// TIA Portal V16 export
// export: Created 2022-11-17T15:49:44.5992417Z, ExportSetting WithDefaults, DisplayName Totally Integrated Automation Portal, DisplayVersion V16 Update 6, DisplayName TIA Portal Version Control Interface, DisplayVersion V16 Update 2, DisplayName TIA Portal Openness, DisplayVersion V16 Update 6, DisplayName SINAMICS Startdrive Advanced, DisplayVersion V16 Update 5, DisplayName SINAMICS Startdrive G130, G150, S120, S150, SINAMICS MV, S210, DisplayVersion V16 Update 5, DisplayName SINAMICS Startdrive G110M, G120, G120C, G120D, G120P, G115D, DisplayVersion V16 Update 5, DisplayName STEP 7 Professional, DisplayVersion V16 Update 6, DisplayName STEP 7 Safety, DisplayVersion V16, DisplayName WinCC Advanced, DisplayVersion V16 Update 6
DATA_BLOCK "DB241_Program9"   // DB241
{ S7_Optimized_Access := 'FALSE' }
AUTHOR : Robopac
VERSION : 0.0
// stored: AutoNumber false, IsOnlyStoredInLoadMemory false, IsWriteProtectedInAS false
   VAR RETAIN
      Program9 { S7_SetPoint := 'True'} : "DatiProgramma";
   END_VAR
BEGIN
   Program9.Wrapping := TRUE;
   Program9.TopLenght := 500;
   Program9.TopRelease := 0;
   Program9.TopDown := 0;
   Program9.Top := 4;
   Program9.PressurePTime := 0;
   Program9.LifterTime := 0;
   Program9.RevOverContrast := 1;
   Program9.RopeEndCycle := 16#02;
   Program9.Spare4 := 16#01;
   Program9.RopeTime := 1500;
   Program9.RevOverClamp := 1;
   Program9.FilmForceFinalRev := 10;
   Program9.FilmPrestretchFinalRev := 100;
   Program9.ArmSpeed := 100;
   Program9.CarriageDown4Top := 500;
   Program9.TopDownTime := 1500;
   Program9.LapsUnderTop := 0;
   Program9.Spare6 := 0;
   Program9.Spare7 := 0;
   Program9.Spare8 := 0;
   Program9.Spare9 := 0;
   Program9.Spare10 := 0;
   Program9.Spare11 := 0;
   Program9.Spare12 := 0;
   Program9.Overlap0_1 := 0;
   Program9.Height1 := 130;
   Program9.Landmark1 := FALSE;
   Program9.Lifter1 := FALSE;
   Program9.SpareBit1H1 := FALSE;
   Program9.Airblower1 := TRUE;
   Program9.NextStep1 := TRUE;
   Program9.PressureP1 := TRUE;
   Program9.SpareByte2H1 := 16#00;
   Program9.Revolution1 := 1;
   Program9.RopeUnit1_1 := 16#01;
   Program9.RopeUnit1_2 := 16#01;
   Program9.FilmForce1 := 5;
   Program9.FilmPrestretch1 := 200;
   Program9.Spare3H1 := 0;
   Program9.Spare49 := 0;
   Program9.Spare50 := 0;
   Program9.Spare51 := 0;
   Program9.Spare52 := 0;
   Program9.Spare53 := 0;
   Program9.Overlap1_2 := 0;
   Program9.Height2 := 50;
   Program9.Landmark2 := FALSE;
   Program9.Lifter2 := FALSE;
   Program9.SpareBit1H2 := FALSE;
   Program9.Airblower2 := TRUE;
   Program9.NextStep2 := TRUE;
   Program9.PressureP2 := TRUE;
   Program9.SpareByte2H2 := 16#00;
   Program9.Revolution2 := 1;
   Program9.RopeUnit2_1 := 16#01;
   Program9.RopeUnit2_2 := 16#01;
   Program9.FilmForce2 := 20;
   Program9.FilmPrestretch2 := 200;
   Program9.Spare3H2 := 0;
   Program9.Spare54 := 0;
   Program9.Spare55 := 0;
   Program9.Spare56 := 0;
   Program9.Spare57 := 0;
   Program9.Spare58 := 0;
   Program9.Overlap2_3 := 100;
   Program9.Height3 := -50;
   Program9.Landmark3 := TRUE;
   Program9.Lifter3 := FALSE;
   Program9.SpareBit1H3 := FALSE;
   Program9.Airblower3 := TRUE;
   Program9.NextStep3 := TRUE;
   Program9.PressureP3 := TRUE;
   Program9.SpareByte2H3 := 16#00;
   Program9.Revolution3 := 2;
   Program9.RopeUnit3_1 := 16#01;
   Program9.RopeUnit3_2 := 16#01;
   Program9.FilmForce3 := 30;
   Program9.FilmPrestretch3 := 200;
   Program9.Spare3H3 := 0;
   Program9.Spare59 := 0;
   Program9.Spare60 := 0;
   Program9.Spare61 := 380;
   Program9.Spare62 := 2800;
   Program9.Spare63 := 0;
   Program9.Overlap3_4 := 100;
   Program9.Height4 := 100;
   Program9.Landmark4 := FALSE;
   Program9.Lifter4 := FALSE;
   Program9.SpareBit1H4 := FALSE;
   Program9.Airblower4 := TRUE;
   Program9.NextStep4 := TRUE;
   Program9.PressureP4 := TRUE;
   Program9.SpareByte2H4 := 16#00;
   Program9.Revolution4 := 3;
   Program9.RopeUnit4_1 := 16#02;
   Program9.RopeUnit4_2 := 16#02;
   Program9.FilmForce4 := 30;
   Program9.FilmPrestretch4 := 200;
   Program9.Spare3H4 := 0;
   Program9.Spare64 := 0;
   Program9.Spare65 := 0;
   Program9.Spare66 := 0;
   Program9.Spare67 := 0;
   Program9.Spare68 := 0;
   Program9.Overlap4_5 := 0;
   Program9.Height5 := 50;
   Program9.Landmark5 := FALSE;
   Program9.Lifter5 := FALSE;
   Program9.SpareBit1H5 := FALSE;
   Program9.Airblower5 := TRUE;
   Program9.NextStep5 := FALSE;
   Program9.PressureP5 := FALSE;
   Program9.SpareByte2H5 := 16#00;
   Program9.Revolution5 := 1;
   Program9.RopeUnit5_1 := 16#01;
   Program9.RopeUnit5_2 := 16#01;
   Program9.FilmForce5 := 30;
   Program9.FilmPrestretch5 := 200;
   Program9.Spare3H5 := 0;
   Program9.Spare69 := 0;
   Program9.Spare70 := 0;
   Program9.Spare71 := 0;
   Program9.Spare72 := 0;
   Program9.Spare73 := 0;
   Program9.Overlap5_6 := 100;
   Program9.Height6 := 50;
   Program9.Landmark6 := FALSE;
   Program9.Lifter6 := FALSE;
   Program9.SpareBit1H6 := FALSE;
   Program9.Airblower6 := TRUE;
   Program9.NextStep6 := FALSE;
   Program9.PressureP6 := FALSE;
   Program9.SpareByte2H6 := 16#00;
   Program9.Revolution6 := 2;
   Program9.RopeUnit6_1 := 16#02;
   Program9.RopeUnit6_2 := 16#01;
   Program9.FilmForce6 := 20;
   Program9.FilmPrestretch6 := 200;
   Program9.Spare3H6 := 0;
   Program9.Spare74 := 0;
   Program9.Spare75 := 0;
   Program9.Spare76 := 0;
   Program9.Spare77 := 0;
   Program9.Spare78 := 0;
   Program9.Overlap6_7 := 0;
   Program9.Height7 := 0;
   Program9.Landmark7 := FALSE;
   Program9.Lifter7 := FALSE;
   Program9.SpareBit1H7 := FALSE;
   Program9.Airblower7 := FALSE;
   Program9.NextStep7 := TRUE;
   Program9.PressureP7 := FALSE;
   Program9.SpareByte2H7 := 16#00;
   Program9.Revolution7 := 1;
   Program9.RopeUnit7_1 := 16#01;
   Program9.RopeUnit7_2 := 16#01;
   Program9.FilmForce7 := 0;
   Program9.FilmPrestretch7 := 100;
   Program9.Spare3H7 := 0;
   Program9.Spare79 := 0;
   Program9.Spare80 := 0;
   Program9.Spare81 := 0;
   Program9.Spare82 := 0;
   Program9.Spare83 := 0;
   Program9.Overlap7_8 := 0;
   Program9.Height8 := 0;
   Program9.Landmark8 := FALSE;
   Program9.Lifter8 := FALSE;
   Program9.SpareBit1H8 := FALSE;
   Program9.Airblower8 := FALSE;
   Program9.NextStep8 := TRUE;
   Program9.PressureP8 := FALSE;
   Program9.SpareByte2H8 := 16#00;
   Program9.Revolution8 := 1;
   Program9.RopeUnit8_1 := 16#01;
   Program9.RopeUnit8_2 := 16#01;
   Program9.FilmForce8 := 0;
   Program9.FilmPrestretch8 := 100;
   Program9.Spare3H8 := 0;
   Program9.Spare84 := 0;
   Program9.Spare85 := 0;
   Program9.Spare86 := 0;
   Program9.Spare87 := 0;
   Program9.Spare88 := 0;
   Program9.Overlap8_9 := 0;
   Program9.Height9 := 0;
   Program9.Landmark9 := FALSE;
   Program9.Lifter9 := FALSE;
   Program9.SpareBit1H9 := FALSE;
   Program9.Airblower9 := FALSE;
   Program9.NextStep9 := TRUE;
   Program9.PressureP9 := FALSE;
   Program9.SpareByte2H9 := 16#00;
   Program9.Revolution9 := 1;
   Program9.RopeUnit9_1 := 16#01;
   Program9.RopeUnit9_2 := 16#01;
   Program9.FilmForce9 := 0;
   Program9.FilmPrestretch9 := 100;
   Program9.Spare3H9 := 0;
   Program9.Spare89 := 0;
   Program9.Spare90 := 0;
   Program9.Spare91 := 0;
   Program9.Spare92 := 0;
   Program9.Spare93 := 0;
   Program9.Overlap9_10 := 0;
   Program9.Height10 := 0;
   Program9.Landmark10 := FALSE;
   Program9.Lifter10 := FALSE;
   Program9.SpareBit1H10 := FALSE;
   Program9.Airblower10 := FALSE;
   Program9.NextStep10 := FALSE;
   Program9.PressureP10 := FALSE;
   Program9.SpareByte2H10 := 16#00;
   Program9.Revolution10 := 1;
   Program9.RopeUnit10_1 := 16#01;
   Program9.RopeUnit10_2 := 16#01;
   Program9.FilmForce10 := 0;
   Program9.FilmPrestretch10 := 100;
   Program9.Spare3H10 := 0;
   Program9.Spare94 := 0;
   Program9.Spare95 := 0;
   Program9.Spare96 := 0;
   Program9.Spare97 := 0;
   Program9.Spare98 := 0;
   Program9.Overlap10_11 := 0;
   Program9.Height11 := 0;
   Program9.Landmark11 := FALSE;
   Program9.Lifter11 := FALSE;
   Program9.SpareBit1H11 := FALSE;
   Program9.Airblower11 := FALSE;
   Program9.NextStep11 := TRUE;
   Program9.PressureP11 := FALSE;
   Program9.SpareByte2H11 := 16#00;
   Program9.Revolution11 := 1;
   Program9.RopeUnit11_1 := 16#01;
   Program9.RopeUnit11_2 := 16#01;
   Program9.FilmForce11 := 0;
   Program9.FilmPrestretch11 := 100;
   Program9.Spare3H11 := 0;
   Program9.Spare99 := 0;
   Program9.Spare100 := 0;
   Program9.Spare101 := 0;
   Program9.Spare102 := 0;
   Program9.Spare103 := 0;
   Program9.Overlap11_12 := 0;
   Program9.Height12 := 0;
   Program9.Landmark12 := FALSE;
   Program9.Lifter12 := FALSE;
   Program9.SpareBit1H12 := FALSE;
   Program9.Airblower12 := FALSE;
   Program9.NextStep12 := FALSE;
   Program9.PressureP12 := FALSE;
   Program9.SpareByte2H12 := 16#00;
   Program9.Revolution12 := 1;
   Program9.RopeUnit12_1 := 16#01;
   Program9.RopeUnit12_2 := 16#01;
   Program9.FilmForce12 := 0;
   Program9.FilmPrestretch12 := 100;
   Program9.Spare3H12 := 0;
   Program9.Spare104 := 0;
   Program9.Spare105 := 0;
   Program9.Spare106 := 0;
   Program9.Spare107 := 0;
   Program9.Spare108 := 0;
END_DATA_BLOCK
